FUNCTION_BLOCK FB_Pump EXTENDS FB_VFD
VAR_INPUT
END_VAR
VAR_OUTPUT
END_VAR
VAR
END_VAR

{warning 'Agregar implementación de método'}
METHOD Scale : BOOL
ScaledAnalog := AnalogSignal * 100;
END_METHOD

END_FUNCTION_BLOCK

(* stored: Version 1.1.0.1, ProductVersion 3.1.4024.12
   POU FB_Pump: Id {8f64b28a-4312-4d8d-8ce7-a7209cc80f47}, SpecialFunc None
   Method Scale: Id {0736ad1e-e81b-44cd-91ae-0b85dc33a765} *)
